// TIA Portal V19 export
ORGANIZATION_BLOCK "Main"   // OB1, LAD, ProgramCycle
TITLE = "Main Program Sweep (Cycle)"
{ S7_Optimized_Access := 'TRUE' }
// stored: SetENOAutomatically false
   VAR_INPUT
      Initial_Call : Bool;   // Initial call of this OB
      Remanence : Bool;   // =True, if remanent data are available
   END_VAR
BEGIN

REGION Network 1: Sensor / States simulation
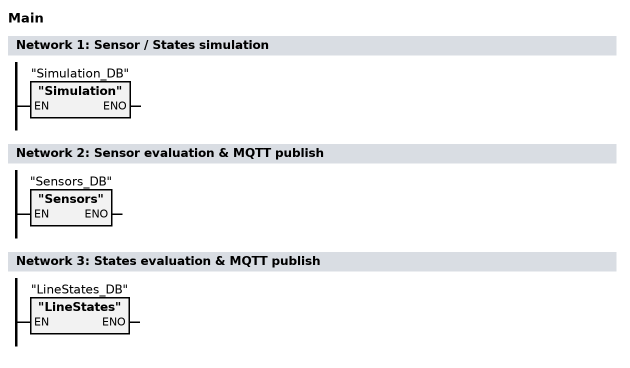
   RUNG wire#powerrail
      "Simulation_DB"()
   END_RUNG
   // the same network as SCL:
   "Simulation_DB"();   // "Simulation"
END_REGION

REGION Network 2: Sensor evaluation & MQTT publish
   RUNG wire#powerrail
      "Sensors_DB"()
   END_RUNG
   // the same network as SCL:
   "Sensors_DB"();   // "Sensors"
END_REGION

REGION Network 3: States evaluation & MQTT publish
   RUNG wire#powerrail
      "LineStates_DB"()
   END_RUNG
   // the same network as SCL:
   "LineStates_DB"();   // "LineStates"
END_REGION
END_ORGANIZATION_BLOCK
